FUNCTION_BLOCK FB_CLAMP
VAR_INPUT
	IN :	BOOL;
	Clamped :	BOOL;
	LimitUpDown :	BOOL;
	VisiSensor :	WORD;
	AllClear :			BOOL; 	//"All clear" -message from picker
END_VAR
VAR_OUTPUT
	Q : 		BOOL;
	StopBlade :	BOOL;
	Clamp :		BOOL;
	Raise :		BOOL;
	ReadyForPickUp: BOOL;
END_VAR
VAR
	iState: INT;
	fbTON: TON;
END_VAR

IF NOT IN THEN
	Q := FALSE;
	iState := 0;
	ELSE
		Q := TRUE;	
END_IF

CASE iState OF
	0 : //idle
	IF Q THEN
		iState := 10;
	END_IF
	10 : //wait for something to CLAMP
	IF VisiSensor = 0 THEN
		StopBlade := FALSE;
		ReadyForPickUp := FALSE;
		ELSE
			StopBlade := TRUE;
			iState := 20;
	END_IF
	20 : //CLAMP CLAMP CLAMP!
	fbTON(IN := TRUE, PT := T#500MS);
	IF fbTON.Q THEN fbTON(IN := FALSE);
		Clamp := TRUE;
		iState := 30;
	END_IF
	30 : //UNCLAMP
	IF Clamped THEN
		Clamp := FALSE;
		iState := 40;
		ReadyForPickUp := TRUE;
	END_IF
	40 : //Wait for all clear
	fbTON(IN := TRUE, PT := T#300MS);
	IF AllClear AND fbTON.Q THEN fbTON(IN := FALSE);
			StopBlade := FALSE;
			iState := 10;
	END_IF
	
END_CASE

END_FUNCTION_BLOCK

(* stored: Version 1.1.0.1, ProductVersion 3.1.4024.6
   POU FB_CLAMP: Id {474c8400-8db1-463b-bf1e-da36c9477ff9}, SpecialFunc None *)
